// TIA Portal V20 export
DATA_BLOCK "LBP_SpindleTempSensor"   // DB1002
TITLE = Spindle temperature sensors / Sondes thermométriques de broche
{ S7_Optimized_Access := 'FALSE' }
AUTHOR : SINUMERIK
FAMILY : SINUMERIK_ONE
VERSION : 6.24
// Interface between user program and operating software, contains signals for spindle temperature sensors / Interface entre programme utilisateur et logiciel d'exploitation, contient des signaux pour sondes thermométriques de broche
// stored: AutoNumber false
   VAR RETAIN
      Sp : Array[1..2] of Struct   // Spindle / Broche
         TS : Array[1..6] of Struct   // Temperature sensor / Sonde thermométrique
            MountPlace : Int;   // Sensor assembly location / Emplacement du module capteur
            Res1 : Int;
            ActVal : Real;   // Temperature sensor actual value [°C] / Sonde thermométrique valeur réelle [°C]
            WarnThreshold : Real;   // Temperature sensor warning threshold value [°C] / Sonde thermométrique valeur seuil d'alarme
            WarnNumLimitViol : Int;   // Number of warning threshold value violations / Nombre de dépassements de la valeur seuil d'alarme
            WarnTsViolYY : Byte;   // Last warning threshold value violation: year / Dernier dépassement de la valeur seuil d'alarme : année
            WarnTsViolMM : Byte;   // Last warning threshold value violation: month / Dernier dépassement de la valeur seuil d'alarme : mois
            WarnTsViolDD : Byte;   // Last warning threshold value violation: day / Dernier dépassement de la valeur seuil d'alarme : jour
            WarnTsViolH : Byte;   // Last warning threshold value violation: hour / Dernier dépassement de la valeur seuil d'alarme : heure
            WarnTsViolM : Byte;   // Last warning threshold value violation: minute / Dernier dépassement de la valeur seuil d'alarme : minute
            WarnTsViolS : Byte;   // Last warning threshold value violation: second / Dernier dépassement de la valeur seuil d'alarme : seconde
            WarnDurLimitViol : DInt;   // Duration of warning threshold value violations / Durée de dépassement de la valeur seuil d'alarme
            FaultThreshold : Real;   // Temperature sensor fault threshold value [°C] / Sonde thermométrique valeur seuil de défaut
            FaultNumLimitViol : Int;   // Number of fault threshold value violations / Nombre de dépassements de la valeur seuil de défaut
            FaultTsViolYY : Byte;   // Last fault threshold value violation: year / Dernier dépassement de la valeur seuil de défaut : année
            FaultTsViolMM : Byte;   // Last fault threshold value violation: month / Dernier dépassement de la valeur seuil de défaut : mois
            FaultTsViolDD : Byte;   // Last fault threshold value violation: day / Dernier dépassement de la valeur seuil de défaut : jour
            FaultTsViolH : Byte;   // Last fault threshold value violation: hour / Dernier dépassement de la valeur seuil de défaut : heure
            FaultTsViolM : Byte;   // Last fault threshold value violation: minute / Dernier dépassement de la valeur seuil de défaut : minute
            FaultTsViolS : Byte;   // Last fault threshold value violation: second / Dernier dépassement de la valeur seuil de défaut : seconde
            FaultDurLimitViol : DInt;   // Duration of fault threshold value violations / Durée de dépassement de la valeur seuil de défaut
         END_STRUCT;
      END_STRUCT;
   END_VAR
BEGIN
   // Sp[1].TS[2].MountPlace : Sensor assembly location / Emplacement du module capteur
   // Sp[1].TS[3].MountPlace : Sensor assembly location / Emplacement du module capteur
   // Sp[1].TS[4].MountPlace : Sensor assembly location / Emplacement du module capteur
   // Sp[1].TS[5].MountPlace : Sensor assembly location / Emplacement du module capteur
   // Sp[1].TS[6].MountPlace : Sensor assembly location / Emplacement du module capteur
   // Sp[2].TS[1].MountPlace : Sensor assembly location / Emplacement du module capteur
   // Sp[2].TS[2].MountPlace : Sensor assembly location / Emplacement du module capteur
   // Sp[2].TS[3].MountPlace : Sensor assembly location / Emplacement du module capteur
   // Sp[2].TS[4].MountPlace : Sensor assembly location / Emplacement du module capteur
   // Sp[2].TS[5].MountPlace : Sensor assembly location / Emplacement du module capteur
   // Sp[2].TS[6].MountPlace : Sensor assembly location / Emplacement du module capteur
   // Sp[1].TS[2].ActVal : Temperature sensor actual value [°C] / Sonde thermométrique valeur réelle [°C]
   // Sp[1].TS[3].ActVal : Temperature sensor actual value [°C] / Sonde thermométrique valeur réelle [°C]
   // Sp[1].TS[4].ActVal : Temperature sensor actual value [°C] / Sonde thermométrique valeur réelle [°C]
   // Sp[1].TS[5].ActVal : Temperature sensor actual value [°C] / Sonde thermométrique valeur réelle [°C]
   // Sp[1].TS[6].ActVal : Temperature sensor actual value [°C] / Sonde thermométrique valeur réelle [°C]
   // Sp[2].TS[1].ActVal : Temperature sensor actual value [°C] / Sonde thermométrique valeur réelle [°C]
   // Sp[2].TS[2].ActVal : Temperature sensor actual value [°C] / Sonde thermométrique valeur réelle [°C]
   // Sp[2].TS[3].ActVal : Temperature sensor actual value [°C] / Sonde thermométrique valeur réelle [°C]
   // Sp[2].TS[4].ActVal : Temperature sensor actual value [°C] / Sonde thermométrique valeur réelle [°C]
   // Sp[2].TS[5].ActVal : Temperature sensor actual value [°C] / Sonde thermométrique valeur réelle [°C]
   // Sp[2].TS[6].ActVal : Temperature sensor actual value [°C] / Sonde thermométrique valeur réelle [°C]
   // Sp[1].TS[2].WarnThreshold : Temperature sensor warning threshold value [°C] / Sonde thermométrique valeur seuil d'alarme
   // Sp[1].TS[3].WarnThreshold : Temperature sensor warning threshold value [°C] / Sonde thermométrique valeur seuil d'alarme
   // Sp[1].TS[4].WarnThreshold : Temperature sensor warning threshold value [°C] / Sonde thermométrique valeur seuil d'alarme
   // Sp[1].TS[5].WarnThreshold : Temperature sensor warning threshold value [°C] / Sonde thermométrique valeur seuil d'alarme
   // Sp[1].TS[6].WarnThreshold : Temperature sensor warning threshold value [°C] / Sonde thermométrique valeur seuil d'alarme
   // Sp[2].TS[1].WarnThreshold : Temperature sensor warning threshold value [°C] / Sonde thermométrique valeur seuil d'alarme
   // Sp[2].TS[2].WarnThreshold : Temperature sensor warning threshold value [°C] / Sonde thermométrique valeur seuil d'alarme
   // Sp[2].TS[3].WarnThreshold : Temperature sensor warning threshold value [°C] / Sonde thermométrique valeur seuil d'alarme
   // Sp[2].TS[4].WarnThreshold : Temperature sensor warning threshold value [°C] / Sonde thermométrique valeur seuil d'alarme
   // Sp[2].TS[5].WarnThreshold : Temperature sensor warning threshold value [°C] / Sonde thermométrique valeur seuil d'alarme
   // Sp[2].TS[6].WarnThreshold : Temperature sensor warning threshold value [°C] / Sonde thermométrique valeur seuil d'alarme
   // Sp[1].TS[2].WarnNumLimitViol : Number of warning threshold value violations / Nombre de dépassements de la valeur seuil d'alarme
   // Sp[1].TS[3].WarnNumLimitViol : Number of warning threshold value violations / Nombre de dépassements de la valeur seuil d'alarme
   // Sp[1].TS[4].WarnNumLimitViol : Number of warning threshold value violations / Nombre de dépassements de la valeur seuil d'alarme
   // Sp[1].TS[5].WarnNumLimitViol : Number of warning threshold value violations / Nombre de dépassements de la valeur seuil d'alarme
   // Sp[1].TS[6].WarnNumLimitViol : Number of warning threshold value violations / Nombre de dépassements de la valeur seuil d'alarme
   // Sp[2].TS[1].WarnNumLimitViol : Number of warning threshold value violations / Nombre de dépassements de la valeur seuil d'alarme
   // Sp[2].TS[2].WarnNumLimitViol : Number of warning threshold value violations / Nombre de dépassements de la valeur seuil d'alarme
   // Sp[2].TS[3].WarnNumLimitViol : Number of warning threshold value violations / Nombre de dépassements de la valeur seuil d'alarme
   // Sp[2].TS[4].WarnNumLimitViol : Number of warning threshold value violations / Nombre de dépassements de la valeur seuil d'alarme
   // Sp[2].TS[5].WarnNumLimitViol : Number of warning threshold value violations / Nombre de dépassements de la valeur seuil d'alarme
   // Sp[2].TS[6].WarnNumLimitViol : Number of warning threshold value violations / Nombre de dépassements de la valeur seuil d'alarme
   // Sp[1].TS[2].WarnTsViolYY : Last warning threshold value violation: year / Dernier dépassement de la valeur seuil d'alarme : année
   // Sp[1].TS[3].WarnTsViolYY : Last warning threshold value violation: year / Dernier dépassement de la valeur seuil d'alarme : année
   // Sp[1].TS[4].WarnTsViolYY : Last warning threshold value violation: year / Dernier dépassement de la valeur seuil d'alarme : année
   // Sp[1].TS[5].WarnTsViolYY : Last warning threshold value violation: year / Dernier dépassement de la valeur seuil d'alarme : année
   // Sp[1].TS[6].WarnTsViolYY : Last warning threshold value violation: year / Dernier dépassement de la valeur seuil d'alarme : année
   // Sp[2].TS[1].WarnTsViolYY : Last warning threshold value violation: year / Dernier dépassement de la valeur seuil d'alarme : année
   // Sp[2].TS[2].WarnTsViolYY : Last warning threshold value violation: year / Dernier dépassement de la valeur seuil d'alarme : année
   // Sp[2].TS[3].WarnTsViolYY : Last warning threshold value violation: year / Dernier dépassement de la valeur seuil d'alarme : année
   // Sp[2].TS[4].WarnTsViolYY : Last warning threshold value violation: year / Dernier dépassement de la valeur seuil d'alarme : année
   // Sp[2].TS[5].WarnTsViolYY : Last warning threshold value violation: year / Dernier dépassement de la valeur seuil d'alarme : année
   // Sp[2].TS[6].WarnTsViolYY : Last warning threshold value violation: year / Dernier dépassement de la valeur seuil d'alarme : année
   // Sp[1].TS[2].WarnTsViolMM : Last warning threshold value violation: month / Dernier dépassement de la valeur seuil d'alarme : mois
   // Sp[1].TS[3].WarnTsViolMM : Last warning threshold value violation: month / Dernier dépassement de la valeur seuil d'alarme : mois
   // Sp[1].TS[4].WarnTsViolMM : Last warning threshold value violation: month / Dernier dépassement de la valeur seuil d'alarme : mois
   // Sp[1].TS[5].WarnTsViolMM : Last warning threshold value violation: month / Dernier dépassement de la valeur seuil d'alarme : mois
   // Sp[1].TS[6].WarnTsViolMM : Last warning threshold value violation: month / Dernier dépassement de la valeur seuil d'alarme : mois
   // Sp[2].TS[1].WarnTsViolMM : Last warning threshold value violation: month / Dernier dépassement de la valeur seuil d'alarme : mois
   // Sp[2].TS[2].WarnTsViolMM : Last warning threshold value violation: month / Dernier dépassement de la valeur seuil d'alarme : mois
   // Sp[2].TS[3].WarnTsViolMM : Last warning threshold value violation: month / Dernier dépassement de la valeur seuil d'alarme : mois
   // Sp[2].TS[4].WarnTsViolMM : Last warning threshold value violation: month / Dernier dépassement de la valeur seuil d'alarme : mois
   // Sp[2].TS[5].WarnTsViolMM : Last warning threshold value violation: month / Dernier dépassement de la valeur seuil d'alarme : mois
   // Sp[2].TS[6].WarnTsViolMM : Last warning threshold value violation: month / Dernier dépassement de la valeur seuil d'alarme : mois
   // Sp[1].TS[2].WarnTsViolDD : Last warning threshold value violation: day / Dernier dépassement de la valeur seuil d'alarme : jour
   // Sp[1].TS[3].WarnTsViolDD : Last warning threshold value violation: day / Dernier dépassement de la valeur seuil d'alarme : jour
   // Sp[1].TS[4].WarnTsViolDD : Last warning threshold value violation: day / Dernier dépassement de la valeur seuil d'alarme : jour
   // Sp[1].TS[5].WarnTsViolDD : Last warning threshold value violation: day / Dernier dépassement de la valeur seuil d'alarme : jour
   // Sp[1].TS[6].WarnTsViolDD : Last warning threshold value violation: day / Dernier dépassement de la valeur seuil d'alarme : jour
   // Sp[2].TS[1].WarnTsViolDD : Last warning threshold value violation: day / Dernier dépassement de la valeur seuil d'alarme : jour
   // Sp[2].TS[2].WarnTsViolDD : Last warning threshold value violation: day / Dernier dépassement de la valeur seuil d'alarme : jour
   // Sp[2].TS[3].WarnTsViolDD : Last warning threshold value violation: day / Dernier dépassement de la valeur seuil d'alarme : jour
   // Sp[2].TS[4].WarnTsViolDD : Last warning threshold value violation: day / Dernier dépassement de la valeur seuil d'alarme : jour
   // Sp[2].TS[5].WarnTsViolDD : Last warning threshold value violation: day / Dernier dépassement de la valeur seuil d'alarme : jour
   // Sp[2].TS[6].WarnTsViolDD : Last warning threshold value violation: day / Dernier dépassement de la valeur seuil d'alarme : jour
   // Sp[1].TS[2].WarnTsViolH : Last warning threshold value violation: hour / Dernier dépassement de la valeur seuil d'alarme : heure
   // Sp[1].TS[3].WarnTsViolH : Last warning threshold value violation: hour / Dernier dépassement de la valeur seuil d'alarme : heure
   // Sp[1].TS[4].WarnTsViolH : Last warning threshold value violation: hour / Dernier dépassement de la valeur seuil d'alarme : heure
   // Sp[1].TS[5].WarnTsViolH : Last warning threshold value violation: hour / Dernier dépassement de la valeur seuil d'alarme : heure
   // Sp[1].TS[6].WarnTsViolH : Last warning threshold value violation: hour / Dernier dépassement de la valeur seuil d'alarme : heure
   // Sp[2].TS[1].WarnTsViolH : Last warning threshold value violation: hour / Dernier dépassement de la valeur seuil d'alarme : heure
   // Sp[2].TS[2].WarnTsViolH : Last warning threshold value violation: hour / Dernier dépassement de la valeur seuil d'alarme : heure
   // Sp[2].TS[3].WarnTsViolH : Last warning threshold value violation: hour / Dernier dépassement de la valeur seuil d'alarme : heure
   // Sp[2].TS[4].WarnTsViolH : Last warning threshold value violation: hour / Dernier dépassement de la valeur seuil d'alarme : heure
   // Sp[2].TS[5].WarnTsViolH : Last warning threshold value violation: hour / Dernier dépassement de la valeur seuil d'alarme : heure
   // Sp[2].TS[6].WarnTsViolH : Last warning threshold value violation: hour / Dernier dépassement de la valeur seuil d'alarme : heure
   // Sp[1].TS[2].WarnTsViolM : Last warning threshold value violation: minute / Dernier dépassement de la valeur seuil d'alarme : minute
   // Sp[1].TS[3].WarnTsViolM : Last warning threshold value violation: minute / Dernier dépassement de la valeur seuil d'alarme : minute
   // Sp[1].TS[4].WarnTsViolM : Last warning threshold value violation: minute / Dernier dépassement de la valeur seuil d'alarme : minute
   // Sp[1].TS[5].WarnTsViolM : Last warning threshold value violation: minute / Dernier dépassement de la valeur seuil d'alarme : minute
   // Sp[1].TS[6].WarnTsViolM : Last warning threshold value violation: minute / Dernier dépassement de la valeur seuil d'alarme : minute
   // Sp[2].TS[1].WarnTsViolM : Last warning threshold value violation: minute / Dernier dépassement de la valeur seuil d'alarme : minute
   // Sp[2].TS[2].WarnTsViolM : Last warning threshold value violation: minute / Dernier dépassement de la valeur seuil d'alarme : minute
   // Sp[2].TS[3].WarnTsViolM : Last warning threshold value violation: minute / Dernier dépassement de la valeur seuil d'alarme : minute
   // Sp[2].TS[4].WarnTsViolM : Last warning threshold value violation: minute / Dernier dépassement de la valeur seuil d'alarme : minute
   // Sp[2].TS[5].WarnTsViolM : Last warning threshold value violation: minute / Dernier dépassement de la valeur seuil d'alarme : minute
   // Sp[2].TS[6].WarnTsViolM : Last warning threshold value violation: minute / Dernier dépassement de la valeur seuil d'alarme : minute
   // Sp[1].TS[2].WarnTsViolS : Last warning threshold value violation: second / Dernier dépassement de la valeur seuil d'alarme : seconde
   // Sp[1].TS[3].WarnTsViolS : Last warning threshold value violation: second / Dernier dépassement de la valeur seuil d'alarme : seconde
   // Sp[1].TS[4].WarnTsViolS : Last warning threshold value violation: second / Dernier dépassement de la valeur seuil d'alarme : seconde
   // Sp[1].TS[5].WarnTsViolS : Last warning threshold value violation: second / Dernier dépassement de la valeur seuil d'alarme : seconde
   // Sp[1].TS[6].WarnTsViolS : Last warning threshold value violation: second / Dernier dépassement de la valeur seuil d'alarme : seconde
   // Sp[2].TS[1].WarnTsViolS : Last warning threshold value violation: second / Dernier dépassement de la valeur seuil d'alarme : seconde
   // Sp[2].TS[2].WarnTsViolS : Last warning threshold value violation: second / Dernier dépassement de la valeur seuil d'alarme : seconde
   // Sp[2].TS[3].WarnTsViolS : Last warning threshold value violation: second / Dernier dépassement de la valeur seuil d'alarme : seconde
   // Sp[2].TS[4].WarnTsViolS : Last warning threshold value violation: second / Dernier dépassement de la valeur seuil d'alarme : seconde
   // Sp[2].TS[5].WarnTsViolS : Last warning threshold value violation: second / Dernier dépassement de la valeur seuil d'alarme : seconde
   // Sp[2].TS[6].WarnTsViolS : Last warning threshold value violation: second / Dernier dépassement de la valeur seuil d'alarme : seconde
   // Sp[1].TS[2].WarnDurLimitViol : Duration of warning threshold value violations / Durée de dépassement de la valeur seuil d'alarme
   // Sp[1].TS[3].WarnDurLimitViol : Duration of warning threshold value violations / Durée de dépassement de la valeur seuil d'alarme
   // Sp[1].TS[4].WarnDurLimitViol : Duration of warning threshold value violations / Durée de dépassement de la valeur seuil d'alarme
   // Sp[1].TS[5].WarnDurLimitViol : Duration of warning threshold value violations / Durée de dépassement de la valeur seuil d'alarme
   // Sp[1].TS[6].WarnDurLimitViol : Duration of warning threshold value violations / Durée de dépassement de la valeur seuil d'alarme
   // Sp[2].TS[1].WarnDurLimitViol : Duration of warning threshold value violations / Durée de dépassement de la valeur seuil d'alarme
   // Sp[2].TS[2].WarnDurLimitViol : Duration of warning threshold value violations / Durée de dépassement de la valeur seuil d'alarme
   // Sp[2].TS[3].WarnDurLimitViol : Duration of warning threshold value violations / Durée de dépassement de la valeur seuil d'alarme
   // Sp[2].TS[4].WarnDurLimitViol : Duration of warning threshold value violations / Durée de dépassement de la valeur seuil d'alarme
   // Sp[2].TS[5].WarnDurLimitViol : Duration of warning threshold value violations / Durée de dépassement de la valeur seuil d'alarme
   // Sp[2].TS[6].WarnDurLimitViol : Duration of warning threshold value violations / Durée de dépassement de la valeur seuil d'alarme
   // Sp[1].TS[2].FaultThreshold : Temperature sensor fault threshold value [°C] / Sonde thermométrique valeur seuil de défaut
   // Sp[1].TS[3].FaultThreshold : Temperature sensor fault threshold value [°C] / Sonde thermométrique valeur seuil de défaut
   // Sp[1].TS[4].FaultThreshold : Temperature sensor fault threshold value [°C] / Sonde thermométrique valeur seuil de défaut
   // Sp[1].TS[5].FaultThreshold : Temperature sensor fault threshold value [°C] / Sonde thermométrique valeur seuil de défaut
   // Sp[1].TS[6].FaultThreshold : Temperature sensor fault threshold value [°C] / Sonde thermométrique valeur seuil de défaut
   // Sp[2].TS[1].FaultThreshold : Temperature sensor fault threshold value [°C] / Sonde thermométrique valeur seuil de défaut
   // Sp[2].TS[2].FaultThreshold : Temperature sensor fault threshold value [°C] / Sonde thermométrique valeur seuil de défaut
   // Sp[2].TS[3].FaultThreshold : Temperature sensor fault threshold value [°C] / Sonde thermométrique valeur seuil de défaut
   // Sp[2].TS[4].FaultThreshold : Temperature sensor fault threshold value [°C] / Sonde thermométrique valeur seuil de défaut
   // Sp[2].TS[5].FaultThreshold : Temperature sensor fault threshold value [°C] / Sonde thermométrique valeur seuil de défaut
   // Sp[2].TS[6].FaultThreshold : Temperature sensor fault threshold value [°C] / Sonde thermométrique valeur seuil de défaut
   // Sp[1].TS[2].FaultNumLimitViol : Number of fault threshold value violations / Nombre de dépassements de la valeur seuil de défaut
   // Sp[1].TS[3].FaultNumLimitViol : Number of fault threshold value violations / Nombre de dépassements de la valeur seuil de défaut
   // Sp[1].TS[4].FaultNumLimitViol : Number of fault threshold value violations / Nombre de dépassements de la valeur seuil de défaut
   // Sp[1].TS[5].FaultNumLimitViol : Number of fault threshold value violations / Nombre de dépassements de la valeur seuil de défaut
   // Sp[1].TS[6].FaultNumLimitViol : Number of fault threshold value violations / Nombre de dépassements de la valeur seuil de défaut
   // Sp[2].TS[1].FaultNumLimitViol : Number of fault threshold value violations / Nombre de dépassements de la valeur seuil de défaut
   // Sp[2].TS[2].FaultNumLimitViol : Number of fault threshold value violations / Nombre de dépassements de la valeur seuil de défaut
   // Sp[2].TS[3].FaultNumLimitViol : Number of fault threshold value violations / Nombre de dépassements de la valeur seuil de défaut
   // Sp[2].TS[4].FaultNumLimitViol : Number of fault threshold value violations / Nombre de dépassements de la valeur seuil de défaut
   // Sp[2].TS[5].FaultNumLimitViol : Number of fault threshold value violations / Nombre de dépassements de la valeur seuil de défaut
   // Sp[2].TS[6].FaultNumLimitViol : Number of fault threshold value violations / Nombre de dépassements de la valeur seuil de défaut
   // Sp[1].TS[2].FaultTsViolYY : Last fault threshold value violation: year / Dernier dépassement de la valeur seuil de défaut : année
   // Sp[1].TS[3].FaultTsViolYY : Last fault threshold value violation: year / Dernier dépassement de la valeur seuil de défaut : année
   // Sp[1].TS[4].FaultTsViolYY : Last fault threshold value violation: year / Dernier dépassement de la valeur seuil de défaut : année
   // Sp[1].TS[5].FaultTsViolYY : Last fault threshold value violation: year / Dernier dépassement de la valeur seuil de défaut : année
   // Sp[1].TS[6].FaultTsViolYY : Last fault threshold value violation: year / Dernier dépassement de la valeur seuil de défaut : année
   // Sp[2].TS[1].FaultTsViolYY : Last fault threshold value violation: year / Dernier dépassement de la valeur seuil de défaut : année
   // Sp[2].TS[2].FaultTsViolYY : Last fault threshold value violation: year / Dernier dépassement de la valeur seuil de défaut : année
   // Sp[2].TS[3].FaultTsViolYY : Last fault threshold value violation: year / Dernier dépassement de la valeur seuil de défaut : année
   // Sp[2].TS[4].FaultTsViolYY : Last fault threshold value violation: year / Dernier dépassement de la valeur seuil de défaut : année
   // Sp[2].TS[5].FaultTsViolYY : Last fault threshold value violation: year / Dernier dépassement de la valeur seuil de défaut : année
   // Sp[2].TS[6].FaultTsViolYY : Last fault threshold value violation: year / Dernier dépassement de la valeur seuil de défaut : année
   // Sp[1].TS[2].FaultTsViolMM : Last fault threshold value violation: month / Dernier dépassement de la valeur seuil de défaut : mois
   // Sp[1].TS[3].FaultTsViolMM : Last fault threshold value violation: month / Dernier dépassement de la valeur seuil de défaut : mois
   // Sp[1].TS[4].FaultTsViolMM : Last fault threshold value violation: month / Dernier dépassement de la valeur seuil de défaut : mois
   // Sp[1].TS[5].FaultTsViolMM : Last fault threshold value violation: month / Dernier dépassement de la valeur seuil de défaut : mois
   // Sp[1].TS[6].FaultTsViolMM : Last fault threshold value violation: month / Dernier dépassement de la valeur seuil de défaut : mois
   // Sp[2].TS[1].FaultTsViolMM : Last fault threshold value violation: month / Dernier dépassement de la valeur seuil de défaut : mois
   // Sp[2].TS[2].FaultTsViolMM : Last fault threshold value violation: month / Dernier dépassement de la valeur seuil de défaut : mois
   // Sp[2].TS[3].FaultTsViolMM : Last fault threshold value violation: month / Dernier dépassement de la valeur seuil de défaut : mois
   // Sp[2].TS[4].FaultTsViolMM : Last fault threshold value violation: month / Dernier dépassement de la valeur seuil de défaut : mois
   // Sp[2].TS[5].FaultTsViolMM : Last fault threshold value violation: month / Dernier dépassement de la valeur seuil de défaut : mois
   // Sp[2].TS[6].FaultTsViolMM : Last fault threshold value violation: month / Dernier dépassement de la valeur seuil de défaut : mois
   // Sp[1].TS[2].FaultTsViolDD : Last fault threshold value violation: day / Dernier dépassement de la valeur seuil de défaut : jour
   // Sp[1].TS[3].FaultTsViolDD : Last fault threshold value violation: day / Dernier dépassement de la valeur seuil de défaut : jour
   // Sp[1].TS[4].FaultTsViolDD : Last fault threshold value violation: day / Dernier dépassement de la valeur seuil de défaut : jour
   // Sp[1].TS[5].FaultTsViolDD : Last fault threshold value violation: day / Dernier dépassement de la valeur seuil de défaut : jour
   // Sp[1].TS[6].FaultTsViolDD : Last fault threshold value violation: day / Dernier dépassement de la valeur seuil de défaut : jour
   // Sp[2].TS[1].FaultTsViolDD : Last fault threshold value violation: day / Dernier dépassement de la valeur seuil de défaut : jour
   // Sp[2].TS[2].FaultTsViolDD : Last fault threshold value violation: day / Dernier dépassement de la valeur seuil de défaut : jour
   // Sp[2].TS[3].FaultTsViolDD : Last fault threshold value violation: day / Dernier dépassement de la valeur seuil de défaut : jour
   // Sp[2].TS[4].FaultTsViolDD : Last fault threshold value violation: day / Dernier dépassement de la valeur seuil de défaut : jour
   // Sp[2].TS[5].FaultTsViolDD : Last fault threshold value violation: day / Dernier dépassement de la valeur seuil de défaut : jour
   // Sp[2].TS[6].FaultTsViolDD : Last fault threshold value violation: day / Dernier dépassement de la valeur seuil de défaut : jour
   // Sp[1].TS[2].FaultTsViolH : Last fault threshold value violation: hour / Dernier dépassement de la valeur seuil de défaut : heure
   // Sp[1].TS[3].FaultTsViolH : Last fault threshold value violation: hour / Dernier dépassement de la valeur seuil de défaut : heure
   // Sp[1].TS[4].FaultTsViolH : Last fault threshold value violation: hour / Dernier dépassement de la valeur seuil de défaut : heure
   // Sp[1].TS[5].FaultTsViolH : Last fault threshold value violation: hour / Dernier dépassement de la valeur seuil de défaut : heure
   // Sp[1].TS[6].FaultTsViolH : Last fault threshold value violation: hour / Dernier dépassement de la valeur seuil de défaut : heure
   // Sp[2].TS[1].FaultTsViolH : Last fault threshold value violation: hour / Dernier dépassement de la valeur seuil de défaut : heure
   // Sp[2].TS[2].FaultTsViolH : Last fault threshold value violation: hour / Dernier dépassement de la valeur seuil de défaut : heure
   // Sp[2].TS[3].FaultTsViolH : Last fault threshold value violation: hour / Dernier dépassement de la valeur seuil de défaut : heure
   // Sp[2].TS[4].FaultTsViolH : Last fault threshold value violation: hour / Dernier dépassement de la valeur seuil de défaut : heure
   // Sp[2].TS[5].FaultTsViolH : Last fault threshold value violation: hour / Dernier dépassement de la valeur seuil de défaut : heure
   // Sp[2].TS[6].FaultTsViolH : Last fault threshold value violation: hour / Dernier dépassement de la valeur seuil de défaut : heure
   // Sp[1].TS[2].FaultTsViolM : Last fault threshold value violation: minute / Dernier dépassement de la valeur seuil de défaut : minute
   // Sp[1].TS[3].FaultTsViolM : Last fault threshold value violation: minute / Dernier dépassement de la valeur seuil de défaut : minute
   // Sp[1].TS[4].FaultTsViolM : Last fault threshold value violation: minute / Dernier dépassement de la valeur seuil de défaut : minute
   // Sp[1].TS[5].FaultTsViolM : Last fault threshold value violation: minute / Dernier dépassement de la valeur seuil de défaut : minute
   // Sp[1].TS[6].FaultTsViolM : Last fault threshold value violation: minute / Dernier dépassement de la valeur seuil de défaut : minute
   // Sp[2].TS[1].FaultTsViolM : Last fault threshold value violation: minute / Dernier dépassement de la valeur seuil de défaut : minute
   // Sp[2].TS[2].FaultTsViolM : Last fault threshold value violation: minute / Dernier dépassement de la valeur seuil de défaut : minute
   // Sp[2].TS[3].FaultTsViolM : Last fault threshold value violation: minute / Dernier dépassement de la valeur seuil de défaut : minute
   // Sp[2].TS[4].FaultTsViolM : Last fault threshold value violation: minute / Dernier dépassement de la valeur seuil de défaut : minute
   // Sp[2].TS[5].FaultTsViolM : Last fault threshold value violation: minute / Dernier dépassement de la valeur seuil de défaut : minute
   // Sp[2].TS[6].FaultTsViolM : Last fault threshold value violation: minute / Dernier dépassement de la valeur seuil de défaut : minute
   // Sp[1].TS[2].FaultTsViolS : Last fault threshold value violation: second / Dernier dépassement de la valeur seuil de défaut : seconde
   // Sp[1].TS[3].FaultTsViolS : Last fault threshold value violation: second / Dernier dépassement de la valeur seuil de défaut : seconde
   // Sp[1].TS[4].FaultTsViolS : Last fault threshold value violation: second / Dernier dépassement de la valeur seuil de défaut : seconde
   // Sp[1].TS[5].FaultTsViolS : Last fault threshold value violation: second / Dernier dépassement de la valeur seuil de défaut : seconde
   // Sp[1].TS[6].FaultTsViolS : Last fault threshold value violation: second / Dernier dépassement de la valeur seuil de défaut : seconde
   // Sp[2].TS[1].FaultTsViolS : Last fault threshold value violation: second / Dernier dépassement de la valeur seuil de défaut : seconde
   // Sp[2].TS[2].FaultTsViolS : Last fault threshold value violation: second / Dernier dépassement de la valeur seuil de défaut : seconde
   // Sp[2].TS[3].FaultTsViolS : Last fault threshold value violation: second / Dernier dépassement de la valeur seuil de défaut : seconde
   // Sp[2].TS[4].FaultTsViolS : Last fault threshold value violation: second / Dernier dépassement de la valeur seuil de défaut : seconde
   // Sp[2].TS[5].FaultTsViolS : Last fault threshold value violation: second / Dernier dépassement de la valeur seuil de défaut : seconde
   // Sp[2].TS[6].FaultTsViolS : Last fault threshold value violation: second / Dernier dépassement de la valeur seuil de défaut : seconde
   // Sp[1].TS[2].FaultDurLimitViol : Duration of fault threshold value violations / Durée de dépassement de la valeur seuil de défaut
   // Sp[1].TS[3].FaultDurLimitViol : Duration of fault threshold value violations / Durée de dépassement de la valeur seuil de défaut
   // Sp[1].TS[4].FaultDurLimitViol : Duration of fault threshold value violations / Durée de dépassement de la valeur seuil de défaut
   // Sp[1].TS[5].FaultDurLimitViol : Duration of fault threshold value violations / Durée de dépassement de la valeur seuil de défaut
   // Sp[1].TS[6].FaultDurLimitViol : Duration of fault threshold value violations / Durée de dépassement de la valeur seuil de défaut
   // Sp[2].TS[1].FaultDurLimitViol : Duration of fault threshold value violations / Durée de dépassement de la valeur seuil de défaut
   // Sp[2].TS[2].FaultDurLimitViol : Duration of fault threshold value violations / Durée de dépassement de la valeur seuil de défaut
   // Sp[2].TS[3].FaultDurLimitViol : Duration of fault threshold value violations / Durée de dépassement de la valeur seuil de défaut
   // Sp[2].TS[4].FaultDurLimitViol : Duration of fault threshold value violations / Durée de dépassement de la valeur seuil de défaut
   // Sp[2].TS[5].FaultDurLimitViol : Duration of fault threshold value violations / Durée de dépassement de la valeur seuil de défaut
   // Sp[2].TS[6].FaultDurLimitViol : Duration of fault threshold value violations / Durée de dépassement de la valeur seuil de défaut
   // Sp[1].TS[1] : Temperature sensor / Sonde thermométrique
   // Sp[1].TS[2] : Temperature sensor / Sonde thermométrique
   // Sp[1].TS[3] : Temperature sensor / Sonde thermométrique
   // Sp[1].TS[4] : Temperature sensor / Sonde thermométrique
   // Sp[1].TS[5] : Temperature sensor / Sonde thermométrique
   // Sp[1].TS[6] : Temperature sensor / Sonde thermométrique
   // Sp[2].TS[1] : Temperature sensor / Sonde thermométrique
   // Sp[2].TS[2] : Temperature sensor / Sonde thermométrique
   // Sp[2].TS[3] : Temperature sensor / Sonde thermométrique
   // Sp[2].TS[4] : Temperature sensor / Sonde thermométrique
   // Sp[2].TS[5] : Temperature sensor / Sonde thermométrique
   // Sp[2].TS[6] : Temperature sensor / Sonde thermométrique
   // Sp[2].TS : Temperature sensor / Sonde thermométrique
   // Sp[1] : Spindle / Broche
   // Sp[2] : Spindle / Broche
END_DATA_BLOCK
